(*
A circular queue implementation for managing `I_Arg`.  
*)
INTERFACE I_MutArgQueue EXTENDS I_ArgQueue

(*
Clears the queue.
*)
METHOD Clear
END_METHOD

(*
Retrieves and removes the next argument from the queue.  
Advances the tail pointer, ensuring cyclic operation within the queue's capacity.
Returns:
- Ok - Returns I_Arg.
- None - Returns null, queue empty.
*)
METHOD Pop : Result
VAR_OUTPUT
	iArg	: I_Arg;
END_VAR
END_METHOD

(*
Adds a new argument to the queue.  
Advances the head pointer while maintaining a cyclic structure, and returns an overflow error if the queue is full.
Returns:
- Ok - Successful insertion
- Err.Ovf - Returns null, the queue is full
*)
METHOD Push : Result
VAR_INPUT
	iArg		: I_Arg;
END_VAR
END_METHOD

END_INTERFACE

(* stored: Version 1.1.0.1
   Itf I_MutArgQueue: Id {3c319922-c4ac-4913-a5ff-e4204e65e323}
   Method Clear: Id {41345009-58c3-4603-a1dd-71a3de823a25}
   Method Pop: Id {be1b5892-95ee-403d-b9ca-f9025d7f85a9}
   Method Push: Id {1f80bd1a-a0b7-40b0-a5e7-7adf8b264e2c} *)
